{attribute 'GeneratedUsingTerminal: EL6201-0000-0017'}
{attribute addProperty BoxType "EL6201-0000-0017"}
{attribute addProperty Id "Slave_5A_DO0BOOL1Slave_5A_DO1BOOL1Slave_5A_DO2BOOL1Slave_5A_DO3BOOL1Slave_5B_DO0BOOL1Slave_5B_DO1BOOL1Slave_5B_DO2BOOL1Slave_5B_DO3BOOL1"}
{attribute addProperty CRC "3986757344"}
{attribute addProperty Size "8"}
TYPE Slave_5_Outputs_EDA116E0 :
STRUCT
	{attribute addProperty Name "Slave_5A_DO0"}
	Slave_5A_DO0 : BOOL;
	{attribute addProperty Name "Slave_5A_DO1"}
	Slave_5A_DO1 : BOOL;
	{attribute addProperty Name "Slave_5A_DO2"}
	Slave_5A_DO2 : BOOL;
	{attribute addProperty Name "Slave_5A_DO3"}
	Slave_5A_DO3 : BOOL;
	{attribute addProperty Name "Slave_5B_DO0"}
	Slave_5B_DO0 : BOOL;
	{attribute addProperty Name "Slave_5B_DO1"}
	Slave_5B_DO1 : BOOL;
	{attribute addProperty Name "Slave_5B_DO2"}
	Slave_5B_DO2 : BOOL;
	{attribute addProperty Name "Slave_5B_DO3"}
	Slave_5B_DO3 : BOOL;
END_STRUCT
END_TYPE

(* stored: Version 1.2.0.0, ProductVersion 3.1.4024.9
   DUT Slave_5_Outputs_EDA116E0: Id {a48ed19c-8685-45b1-994e-834bac073836} *)
